FUNCTION_BLOCK MultiActStatus (* Composite Function Block Type *)
  (* Standard: 61499-2 *)
  (* Version 0.0, 6/9/2026, Schneider Electric, template *)
  PACKAGE SE.Nereda;
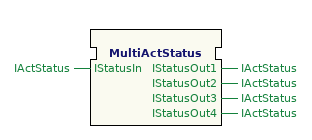
  SOCKETS
    IStatusIn : IActStatus;
  END_SOCKETS
  PLUGS
    IStatusOut1 : IActStatus;
    IStatusOut2 : IActStatus;
    IStatusOut3 : IActStatus;
    IStatusOut4 : IActStatus;
  END_PLUGS
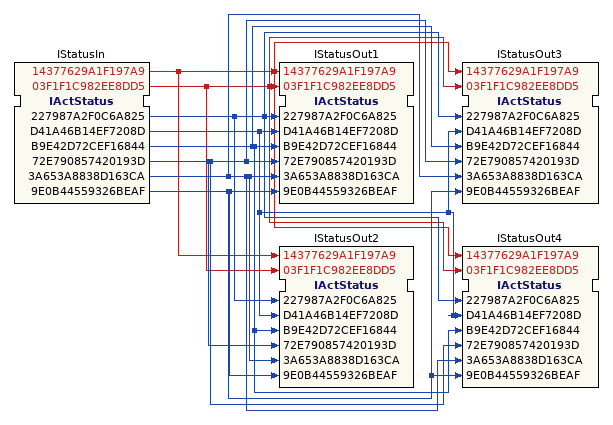
  EVENT_CONNECTIONS
    IStatusIn.14377629A1F197A9 TO IStatusOut1.14377629A1F197A9;
    IStatusIn.14377629A1F197A9 TO IStatusOut3.14377629A1F197A9;
    IStatusIn.14377629A1F197A9 TO IStatusOut2.14377629A1F197A9;
    IStatusIn.14377629A1F197A9 TO IStatusOut4.14377629A1F197A9;
    IStatusIn.03F1F1C982EE8DD5 TO IStatusOut1.03F1F1C982EE8DD5;
    IStatusIn.03F1F1C982EE8DD5 TO IStatusOut3.03F1F1C982EE8DD5;
    IStatusIn.03F1F1C982EE8DD5 TO IStatusOut2.03F1F1C982EE8DD5;
    IStatusIn.03F1F1C982EE8DD5 TO IStatusOut4.03F1F1C982EE8DD5;
  END_CONNECTIONS
  DATA_CONNECTIONS
    IStatusIn.227987A2F0C6A825 TO IStatusOut1.227987A2F0C6A825;
    IStatusIn.227987A2F0C6A825 TO IStatusOut3.227987A2F0C6A825;
    IStatusIn.227987A2F0C6A825 TO IStatusOut2.227987A2F0C6A825;
    IStatusIn.227987A2F0C6A825 TO IStatusOut4.227987A2F0C6A825;
    IStatusIn.D41A46B14EF7208D TO IStatusOut1.D41A46B14EF7208D;
    IStatusIn.D41A46B14EF7208D TO IStatusOut3.D41A46B14EF7208D;
    IStatusIn.D41A46B14EF7208D TO IStatusOut2.D41A46B14EF7208D;
    IStatusIn.D41A46B14EF7208D TO IStatusOut4.D41A46B14EF7208D;
    IStatusIn.B9E42D72CEF16844 TO IStatusOut1.B9E42D72CEF16844;
    IStatusIn.B9E42D72CEF16844 TO IStatusOut3.B9E42D72CEF16844;
    IStatusIn.B9E42D72CEF16844 TO IStatusOut2.B9E42D72CEF16844;
    IStatusIn.B9E42D72CEF16844 TO IStatusOut4.B9E42D72CEF16844;
    IStatusIn.72E790857420193D TO IStatusOut1.72E790857420193D;
    IStatusIn.72E790857420193D TO IStatusOut3.72E790857420193D;
    IStatusIn.72E790857420193D TO IStatusOut2.72E790857420193D;
    IStatusIn.72E790857420193D TO IStatusOut4.72E790857420193D;
    IStatusIn.3A653A8838D163CA TO IStatusOut1.3A653A8838D163CA;
    IStatusIn.3A653A8838D163CA TO IStatusOut3.3A653A8838D163CA;
    IStatusIn.3A653A8838D163CA TO IStatusOut2.3A653A8838D163CA;
    IStatusIn.3A653A8838D163CA TO IStatusOut4.3A653A8838D163CA;
    IStatusIn.9E0B44559326BEAF TO IStatusOut1.9E0B44559326BEAF;
    IStatusIn.9E0B44559326BEAF TO IStatusOut3.9E0B44559326BEAF;
    IStatusIn.9E0B44559326BEAF TO IStatusOut2.9E0B44559326BEAF;
    IStatusIn.9E0B44559326BEAF TO IStatusOut4.9E0B44559326BEAF;
  END_CONNECTIONS
END_FUNCTION_BLOCK
